# EPICS autosave request: ADFireWireWin/firewireWinApp/Db/firewireFeatureAbs_settings.req
$(P)$(R)$(FEATURE)_ABS
$(P)$(R)$(FEATURE)_CTRL
